FUNCTION_BLOCK "LAcycCom_WriteDriveParams"
{ S7_Optimized_Access := 'TRUE' }
AUTHOR : 'tech.team.motioncontrol@siemens.com'
FAMILY : AcycCom
VERSION : 1.5
   VAR_INPUT
      execute : Bool;
      parameterCount : Int := -1;
      driveObjectId { S7_HiddenAssignment := 'HideIfNoParamAssigned'} : Int := -1;
      hardwareId : HW_IO;
   END_VAR

   VAR_OUTPUT
      done { ExternalWritable := 'False'} : Bool;
      busy { ExternalWritable := 'False'} : Bool;
      error { ExternalWritable := 'False'} : Bool;
      status { ExternalWritable := 'False'} : Word := #STATUS_NO_CALL;
      diagnostics { ExternalWritable := 'False'} : "LAcycCom_typeDriveDiagnostics";
   END_VAR

   VAR_IN_OUT
      requestBuffer : "LAcycCom_typeRequestBuffer";
      dataset : Variant;
   END_VAR

   VAR
      statExecuteOld { ExternalAccessible := 'False'; ExternalVisible := 'False'; ExternalWritable := 'False'} : Bool := FALSE;
      statBusy { ExternalAccessible := 'False'; ExternalVisible := 'False'; ExternalWritable := 'False'} : Bool := FALSE;
      statDone { ExternalAccessible := 'False'; ExternalVisible := 'False'; ExternalWritable := 'False'} : Bool := FALSE;
      statError { ExternalAccessible := 'False'; ExternalVisible := 'False'; ExternalWritable := 'False'} : Bool := FALSE;
      statCmdBusy { ExternalAccessible := 'False'; ExternalVisible := 'False'; ExternalWritable := 'False'} : Bool := FALSE;
      statCmdDone { ExternalAccessible := 'False'; ExternalVisible := 'False'; ExternalWritable := 'False'} : Bool := FALSE;
      statCmdError { ExternalAccessible := 'False'; ExternalVisible := 'False'; ExternalWritable := 'False'} : Bool := FALSE;
      statTimerStart { ExternalAccessible := 'False'; ExternalVisible := 'False'; ExternalWritable := 'False'} : Bool := FALSE;
      statDoId { ExternalAccessible := 'False'; ExternalVisible := 'False'; ExternalWritable := 'False'} : Byte := 16#00;
      statHwId { ExternalAccessible := 'False'; ExternalVisible := 'False'; ExternalWritable := 'False'} : HW_IO := 16#0000;
      statRefNo { ExternalAccessible := 'False'; ExternalVisible := 'False'; ExternalWritable := 'False'} : Byte := 16#00;
      statStatus { ExternalAccessible := 'False'; ExternalVisible := 'False'; ExternalWritable := 'False'} : Word := #STATUS_NO_CALL;
      statSubfunctionStatus { ExternalAccessible := 'False'; ExternalVisible := 'False'; ExternalWritable := 'False'} : Word := 16#0000;
      statWithoutResourceManager { ExternalAccessible := 'False'; ExternalVisible := 'False'; ExternalWritable := 'False'} : Bool := FALSE;
      statFBState { ExternalAccessible := 'False'; ExternalVisible := 'False'; ExternalWritable := 'False'} : SInt := #FB_IDLE;
      statFBSubState { ExternalAccessible := 'False'; ExternalVisible := 'False'; ExternalWritable := 'False'} : SInt := #FB_BUSY_WRREC_1;
      statFBSubStateOld { ExternalAccessible := 'False'; ExternalVisible := 'False'; ExternalWritable := 'False'} : SInt := #FB_BUSY_WRREC_1;
      statStateNumber { ExternalAccessible := 'False'; ExternalVisible := 'False'; ExternalWritable := 'False'} : SInt := 0;
      statDatasetType { ExternalAccessible := 'False'; ExternalVisible := 'False'; ExternalWritable := 'False'} : SInt := 0;
      statErrorCount { ExternalAccessible := 'False'; ExternalVisible := 'False'; ExternalWritable := 'False'} : UInt := 16#0000;
      statAllocatedIndex { ExternalAccessible := 'False'; ExternalVisible := 'False'; ExternalWritable := 'False'} : Int := 0;
      statCountOfElements { ExternalAccessible := 'False'; ExternalVisible := 'False'; ExternalWritable := 'False'} : Int := 0;
      statFirstParameterError { ExternalAccessible := 'False'; ExternalVisible := 'False'; ExternalWritable := 'False'} : Int := -1;
      statWarningRetriggering { ExternalAccessible := 'False'; ExternalVisible := 'False'; ExternalWritable := 'False'} : Bool;
      statDataRecordNo { ExternalAccessible := 'False'; ExternalVisible := 'False'; ExternalWritable := 'False'} : DInt;
      statParameter { ExternalAccessible := 'False'; ExternalVisible := 'False'; ExternalWritable := 'False'} : Array[0..#WRITE_PARAMETERS_UPPER_LIM] of Struct
         parameterNo { ExternalAccessible := 'False'; ExternalVisible := 'False'; ExternalWritable := 'False'} : UInt;
         index { ExternalAccessible := 'False'; ExternalVisible := 'False'; ExternalWritable := 'False'} : UInt;
         realValue { ExternalAccessible := 'False'; ExternalVisible := 'False'; ExternalWritable := 'False'} : Real;
         dwordValue { ExternalAccessible := 'False'; ExternalVisible := 'False'; ExternalWritable := 'False'} : DWord;
         format { ExternalAccessible := 'False'; ExternalVisible := 'False'; ExternalWritable := 'False'} : Byte;
         errorValue { ExternalAccessible := 'False'; ExternalVisible := 'False'; ExternalWritable := 'False'} : Byte;
      END_STRUCT;
      statReqReadParameter { ExternalAccessible := 'False'; ExternalVisible := 'False'; ExternalWritable := 'False'} : Struct
         header { ExternalAccessible := 'False'; ExternalVisible := 'False'; ExternalWritable := 'False'} : Struct
            refNo { ExternalAccessible := 'False'; ExternalVisible := 'False'; ExternalWritable := 'False'} : Byte;
            reqId { ExternalAccessible := 'False'; ExternalVisible := 'False'; ExternalWritable := 'False'} : Byte;
            doId { ExternalAccessible := 'False'; ExternalVisible := 'False'; ExternalWritable := 'False'} : Byte;
            parameterNo { ExternalAccessible := 'False'; ExternalVisible := 'False'; ExternalWritable := 'False'} : Byte;
         END_STRUCT;
         parameterAddress { ExternalAccessible := 'False'; ExternalVisible := 'False'; ExternalWritable := 'False'} : Array[0..#WRITE_PARAMETERS_UPPER_LIM] of Struct
            attribute { ExternalAccessible := 'False'; ExternalVisible := 'False'; ExternalWritable := 'False'} : Byte;
            elementNo { ExternalAccessible := 'False'; ExternalVisible := 'False'; ExternalWritable := 'False'} : Byte;
            parameterNo { ExternalAccessible := 'False'; ExternalVisible := 'False'; ExternalWritable := 'False'} : UInt;
            index { ExternalAccessible := 'False'; ExternalVisible := 'False'; ExternalWritable := 'False'} : UInt;
         END_STRUCT;
      END_STRUCT;
      statReqParameterInit { ExternalAccessible := 'False'; ExternalVisible := 'False'; ExternalWritable := 'False'} : Struct
         attribute { ExternalAccessible := 'False'; ExternalVisible := 'False'; ExternalWritable := 'False'} : Byte := 16#10;
         elementNo { ExternalAccessible := 'False'; ExternalVisible := 'False'; ExternalWritable := 'False'} : Byte := 16#01;
         parameterNo { ExternalAccessible := 'False'; ExternalVisible := 'False'; ExternalWritable := 'False'} : UInt := 0;
         index { ExternalAccessible := 'False'; ExternalVisible := 'False'; ExternalWritable := 'False'} : UInt := 0;
      END_STRUCT;
      statReqWriteParameter { ExternalAccessible := 'False'; ExternalVisible := 'False'; ExternalWritable := 'False'} : Struct
         header { ExternalAccessible := 'False'; ExternalVisible := 'False'; ExternalWritable := 'False'} : Struct
            refNo { ExternalAccessible := 'False'; ExternalVisible := 'False'; ExternalWritable := 'False'} : Byte;
            reqId { ExternalAccessible := 'False'; ExternalVisible := 'False'; ExternalWritable := 'False'} : Byte;
            doId { ExternalAccessible := 'False'; ExternalVisible := 'False'; ExternalWritable := 'False'} : Byte;
            parameterNo { ExternalAccessible := 'False'; ExternalVisible := 'False'; ExternalWritable := 'False'} : Byte;
         END_STRUCT;
         data { ExternalAccessible := 'False'; ExternalVisible := 'False'; ExternalWritable := 'False'} : Array[0..#LENGTH_WRITE_TELEGRAM_UPPER_LIM] of Byte;
      END_STRUCT;
      statRespParameter { ExternalAccessible := 'False'; ExternalVisible := 'False'; ExternalWritable := 'False'} : Struct
         header { ExternalAccessible := 'False'; ExternalVisible := 'False'; ExternalWritable := 'False'} : Struct
            refNo { ExternalAccessible := 'False'; ExternalVisible := 'False'; ExternalWritable := 'False'} : Byte;
            reqId { ExternalAccessible := 'False'; ExternalVisible := 'False'; ExternalWritable := 'False'} : Byte;
            doId { ExternalAccessible := 'False'; ExternalVisible := 'False'; ExternalWritable := 'False'} : Byte;
            parameterNo { ExternalAccessible := 'False'; ExternalVisible := 'False'; ExternalWritable := 'False'} : Byte;
         END_STRUCT;
         data { ExternalAccessible := 'False'; ExternalVisible := 'False'; ExternalWritable := 'False'} : Array[0..#LENGTH_READ_TELEGRAM_UPPER_LIM] of Byte;
      END_STRUCT;
      instWRREC {InstructionName := 'WRREC'; LibVersion := '1.1'; ExternalAccessible := 'False'; ExternalVisible := 'False'; ExternalWritable := 'False'} : WRREC;
      instRDREC {InstructionName := 'RDREC'; LibVersion := '1.0'; ExternalAccessible := 'False'; ExternalVisible := 'False'; ExternalWritable := 'False'} : RDREC;
      instIECTimer {InstructionName := 'TON_TIME'; LibVersion := '1.0'; ExternalAccessible := 'False'; ExternalVisible := 'False'; ExternalWritable := 'False'} : TON_TIME;
   END_VAR

   VAR_TEMP
      tempExecute : Bool;
      tempCmdValid : Bool;
      tempStatusWord : Word;
      tempParameterCount : Int;
      tempPointer : Int;
      tempLoopIndex : Int;
      tempBlkVariant : Int;
      tempLastQueueElement : Int;
      tempCmdStatus : DWord;
      tempDWord : DWord;
      tempVoidDiagnostics : "LAcycCom_typeDriveDiagnostics";
      tempActualElementReal : "LAcycCom_typeDriveDatasetReal";
      tempActualElementDWord : "LAcycCom_typeDriveDatasetDWord";
      tempSilentOperationData : "LAcycCom_typeDriveSilentOperation";
      tempVoidHeader : Struct
         reqRef : Byte;
         reqId : Byte;
         axisNo : Byte;
         parameterNo : Byte;
      END_STRUCT;
      tempDatasetRealValue : Array[0..1] of "LAcycCom_typeDriveDatasetReal";
      tempDatasetDWordValue : Array[0..1] of "LAcycCom_typeDriveDatasetDWord";
   END_VAR

   VAR CONSTANT
      DATA_TYPE_SILENT : SInt := 1;
      DATA_TYPE_DATASET_REAL : SInt := 2;
      DATA_TYPE_DATASET_DWORD : SInt := 3;
      NO_PARAMETER_ERROR : Int := -1;
      ALL_ELEMENTS_OCCUPIED : Int := -1;
      FB_IDLE : SInt := 0;
      FB_FIRST_CYCLE : SInt := 1;
      FB_ALLOCATE : SInt := 2;
      FB_GET_RESOURCE : SInt := 3;
      FB_BUSY : SInt := 4;
      FB_RELEASE : SInt := 5;
      FB_DONE : SInt := 6;
      FB_ERROR : SInt := 7;
      FB_BUSY_WRREC_1 : SInt := 8;
      FB_BUSY_WRREC_2 : SInt := 9;
      FB_BUSY_RDREC_1 : SInt := 10;
      FB_BUSY_RDREC_2 : SInt := 11;
      FB_BUSY_WAIT : SInt := 12;
      FORMAT_INTEGER_8 : SInt := 2;
      FORMAT_INTEGER_16 : SInt := 3;
      FORMAT_INTEGER_32 : SInt := 4;
      FORMAT_UNSIGNED_8 : SInt := 5;
      FORMAT_UNSIGNED_16 : SInt := 6;
      FORMAT_UNSIGNED_32 : SInt := 7;
      FORMAT_FLOATING_POINT : SInt := 8;
      FORMAT_OCTET_STRING : SInt := 10;
      FORMAT_TIME_DIFFERENCE : SInt := 13;
      FORMAT_ZERO : SInt := 64;
      FORMAT_BYTE : SInt := 65;
      FORMAT_WORD : SInt := 66;
      FORMAT_DOUBLE_WORD : SInt := 67;
      FORMAT_ERROR : Byte := 16#44;
      WRITE_PARAMETERS_UPPER_LIM : Int := 18;
      SILENT_OPERATION_PARA_UPPER_LIM : Int := 17;
      LENGTH_WRITE_TELEGRAM_UPPER_LIM : Int := 227;
      LENGTH_READ_TELEGRAM_UPPER_LIM : Int := 113;
      MAX_ERROR_COUNT : UInt := 100;
      TIMER_TEMP_ERROR : Time := T#200MS;
      TIMER_ALLOCATION : Time := T#10S;
      MAX_DRIVE_OBJECT_NO : Int := 254;
      STATUS_EXECUTION_FINISHED : Word := 16#0000;
      STATUS_NO_CALL : Word := 16#7000;
      STATUS_ALLOCATE : Word := 16#7001;
      STATUS_GET_RESOURCE : Word := 16#7002;
      STATUS_BUSY : Word := 16#7003;
      STATUS_RELEASE : Word := 16#7004;
      WARN_EXECUTE : Word := 16#7100;
      WARN_EXECUTE_SET_DURING_PROCESSING : Word := 16#7101;
      ERR_NO_OF_PARAMETERS : Word := 16#8001;
      ERR_REQUEST_REJECTED : Word := 16#8004;
      ERR_RESOURCE_RELEASED : Word := 16#8005;
      ERR_AMBIGUOUS_FB_CALL : Word := 16#8006;
      ERR_INVALID_DATA_TYPE : Word := 16#8200;
      ERR_INVALID_BUF_INDEX : Word := 16#8201;
      ERR_INVALID_DRIVE_OBJECT_ID : Word := 16#8208;
      ERR_COMMAND_TIMEOUT : Word := 16#8600;
      ERR_RDREC_TEMP_COUNTER : Word := 16#8601;
      ERR_WRREC_TEMP_COUNTER : Word := 16#8602;
      ERR_WRREC : Word := 16#8603;
      ERR_RDREC : Word := 16#8604;
      ERR_REFERENCE_NO : Word := 16#8605;
      ERR_RESPONSE_ID : Word := 16#8606;
      ERR_PARAMETER_NO : Word := 16#8607;
      ERR_DRIVE_OBJECT_NO : Word := 16#8608;
      ERR_ALLOCATION_TIME : Word := 16#8609;
      ERR_MOVE_BLK_VARIANT : Word := 16#8610;
      ERR_UNDEFINED_STATE : Word := 16#8611;
      ERR_UNDEFINED_SUBSTATE : Word := 16#8612;
      ERR_PARAMETER : Word := 16#8619;
   END_VAR


BEGIN
	//==========================================================================================
	// SIEMENS AG
	// (c)Copyright 2020 All Rights Reserved
	//------------------------------------------------------------------------------------------
	// Library: LAcycCom
	// Tested with: S7-1513-1 PN
	// Engineering: TIA Portal V15
	// Restrictions: ---
	// Requirements: S7-1200/1500
	//               FB LAcycCom_ResourceManager is required
	// Functionality: Writes parameters into a drive object according to the configured dataset
	//------------------------------------------------------------------------------------------
	// Change log table:
	// Version    Date          Expert in charge    Changes applied
	// 01.00.00   05.05.2015    AW                  release
	// 01.01.00   27.01.2016    AW                  values of MAX_ERROR_COUNT and TIMER_TEMP_ERROR changed
	// 01.03.00   05.07.2016    AL                  output added: diagnostics.status
	//                                              bugfix error handling (if execute input is set only for 1 cycle)
	// 01.03.01   21.11.2016    AL                  prevent reentrant calls (added warning #WARN_EXECUTE_SET_DURING_PROCESSING
	//                                                                       and error #ERR_AMBIGUOUS_FB_CALL)
	// 01.03.02   22.11.2017    AL                  added handling of error 80A0 (RDREC)
	//                                              added handling of error 80A1 (WRREC)
	//                                              added errorValue to "LAcycCom_typeDriveDiagnostics"
	// 01.03.03   13.03.2018    AL                  values of MAX_ERROR_COUNT and TIMER_TEMP_ERROR changed
	// 01.05.00   31.10.2018    AL                  added support of Base Mode Parameter Access local (16#B02E)
	//                                              (driveObjectId < 0: local, driveObjectId >= 0: Base Mode Parameter Access global via dataset 47)
	//                                              input 'driveObjectId' data type changed from USInt to Int
	//                                              changed handling of OCTET_STRING format
	// 01.05.01   11.10.2019    AL                  bugfix lockBuffer
	//                                              value of MAX_ERROR_COUNT changed
	// 01.05.02   19.05.2020    CR                  new errorId when input 'driveObjectId' is out of range
	//
	//------------------------------------------------------------------------------------------
	// Function block: LAcycCom_WriteDriveParams
	//===========================================================================================
	//

	//----------------------------------------------------------------------
	// Determine which PLC data type for writeDataset is in use
	//----------------------------------------------------------------------
	IF (TypeOf(#dataset) = TypeOf(#tempDatasetRealValue)) OR (TypeOf(#dataset) = TypeOf(#tempDatasetDWordValue)) THEN
	  #tempExecute := #execute;

	ELSIF (TypeOf(#dataset) = LAcycCom_typeDriveSilentOperation) THEN
	  #tempBlkVariant := MOVE_BLK_VARIANT(SRC := #dataset, COUNT := 1, SRC_INDEX := 0, DEST_INDEX := 0, DEST => #tempSilentOperationData);

	  // Error occurred during MOVE_BLK_VARIANT command
	  IF (#tempBlkVariant <> 0) THEN
	    #statError := TRUE;
	    #statStateNumber := #statFBState;
	    #statSubfunctionStatus := INT_TO_WORD(#tempBlkVariant);
	    #statStatus := #ERR_MOVE_BLK_VARIANT;
	    #statFBState := #FB_ERROR;
	  END_IF;

	  #tempExecute := #tempSilentOperationData.functionBlockCommand.%X1;

	  // Input execute is set during silent operation
	  IF (#execute = TRUE) AND (#statError = FALSE) THEN
	    #statStatus := #WARN_EXECUTE;
	    #diagnostics.status := #statStatus;
	  END_IF;

	ELSE
	  #statError := TRUE;
	  #statStateNumber := #statFBState;
	  #statStatus := #ERR_INVALID_DATA_TYPE;
	  #statFBState := #FB_ERROR;
	END_IF;

	//----------------------------------------------------------------------
	// Processing
	//----------------------------------------------------------------------
	// Rising edge of execute starts functionality
	IF (#tempExecute = TRUE) AND (#statExecuteOld = FALSE) AND (#statBusy = TRUE) THEN
	  // Input execute is set during processing
	  #statStatus := #WARN_EXECUTE_SET_DURING_PROCESSING;
	  #statWarningRetriggering := TRUE;

	ELSIF (#tempExecute = TRUE) AND (#statExecuteOld = FALSE) THEN
	  // First call
	  // Initialisation
	  #statDone := FALSE;
	  #statBusy := TRUE;
	  #statError := FALSE;
	  #statCountOfElements := 0;
	  #statAllocatedIndex := 0;
	  #statHwId := 16#0;
	  #statSubfunctionStatus := 16#0;
	  #statDoId := 0;
	  #statDataRecordNo := 0;
	  #statStateNumber := 0;
	  #statFirstParameterError := -1;
	  #statCmdBusy := FALSE;
	  #statCmdDone := FALSE;
	  #statCmdError := FALSE;
	  #statErrorCount := 0;
	  #statWarningRetriggering := FALSE;
	  #statFBSubState := #FB_BUSY_WRREC_1;
	  #statFBState := #FB_FIRST_CYCLE;

	  #instIECTimer(IN := FALSE,
	                PT := #TIMER_ALLOCATION);

	  // FB is currently inactive
	ELSIF (#tempExecute = FALSE) AND (#statBusy = FALSE)
	THEN
	  #statError := FALSE;
	  #statBusy := FALSE;
	  #statDone := FALSE;
	  #statFBState := #FB_IDLE;

	  IF (#statStatus = #WARN_EXECUTE) AND (#execute = FALSE) OR (#statStatus <> #WARN_EXECUTE) THEN
	    #statStatus := #STATUS_NO_CALL;
	  END_IF;
	END_IF; // #tempExecute AND NOT #statExecuteOld

	//----------------------------------------------------------------------
	// State Machine
	//----------------------------------------------------------------------

	IF (#statBusy = TRUE) AND (#statError = FALSE) THEN  // Functionality running
	  CASE #statFBState OF
	    #FB_FIRST_CYCLE:  // First cycle state

	      // Determine which PLC data type for readDataset is in use
	      IF (TypeOf(#dataset) = TypeOf(#tempDatasetRealValue)) THEN
	        #statDatasetType := #DATA_TYPE_DATASET_REAL;

	      ELSIF (TypeOf(#dataset) = TypeOf(#tempDatasetDWordValue)) THEN
	        #statDatasetType := #DATA_TYPE_DATASET_DWORD;

	      ELSIF (TypeOf(#dataset) = LAcycCom_typeDriveSilentOperation) THEN
	        #statDatasetType := #DATA_TYPE_SILENT;
	      END_IF;

	      // Clearing the dataset in silent operation mode
	      FOR #tempLoopIndex := 0 TO #SILENT_OPERATION_PARA_UPPER_LIM DO
	        #tempSilentOperationData.dataset[#tempLoopIndex].errorValue := 16#FF;
	      END_FOR;

	      // Clearing the sending read buffer
	      #statReqReadParameter.header := #tempVoidHeader;
	      FOR #tempLoopIndex := 0 TO #WRITE_PARAMETERS_UPPER_LIM DO
	        #statReqReadParameter.parameterAddress[#tempLoopIndex] := #statReqParameterInit;
	      END_FOR;

	      // Clearing the sending write buffer
	      #statReqWriteParameter.header := #tempVoidHeader;
	      FOR #tempLoopIndex := 0 TO #LENGTH_WRITE_TELEGRAM_UPPER_LIM DO
	        #statReqWriteParameter.data[#tempLoopIndex] := 16#00;
	      END_FOR;

	      // Clearing the receive buffer
	      #statRespParameter.header := #tempVoidHeader;
	      FOR #tempLoopIndex := 0 TO #LENGTH_READ_TELEGRAM_UPPER_LIM DO
	        #statRespParameter.data[#tempLoopIndex] := 16#00;
	      END_FOR;

	      // Initialization after start, depending on the used PLC data type
	      IF (#statDatasetType = #DATA_TYPE_DATASET_REAL) OR (#statDatasetType = #DATA_TYPE_DATASET_DWORD) THEN
	        IF #driveObjectId < 0 THEN // V1.5
	          #statDataRecordNo := 16#B02E; // Base Mode Parameter Access local; doId not relevant
	          #statDoId := 0;

	        ELSIF (#driveObjectId <= #MAX_DRIVE_OBJECT_NO)
	          AND (#driveObjectId <> 0)
	        THEN // V1.5.2
	          #statDataRecordNo := 47; // Data record 47; Base Mode Parameter Access global
	          #statDoId := INT_TO_BYTE(#driveObjectId);

	        ELSE // V1.5.2
	          // Wrong drive object ID at input
	          #statError := TRUE;
	          #statStateNumber := #statFBState;
	          #statStatus := #ERR_INVALID_DRIVE_OBJECT_ID;
	          #statFBState := #FB_ERROR;
	        END_IF;

	        #statHwId := #hardwareId;
	        #tempParameterCount := #parameterCount;
	      ELSE
	        IF #tempSilentOperationData.driveObjectId < 0 THEN // V1.5
	          #statDataRecordNo := 16#B02E; // Base Mode Parameter Access local; doId not relevant
	          #statDoId := 0;
	        ELSE
	          #statDataRecordNo := 47; // Data record 47; Base Mode Parameter Access global
	          #statDoId := INT_TO_BYTE(#tempSilentOperationData.driveObjectId);
	        END_IF;
	        #statHwId := #tempSilentOperationData.hardwareId;
	        #tempParameterCount := #tempSilentOperationData.parameterCount;
	      END_IF;

	      #diagnostics := #tempVoidDiagnostics;
	      // Input execute is set during silent operation
	      IF #statStatus = #WARN_EXECUTE THEN
	        #diagnostics.status := #statStatus;
	      END_IF;
	      #diagnostics.driveObjectId := #statDoId;
	      #diagnostics.hardwareId := #statHwId;
	      #diagnostics.firstParameterError := #statFirstParameterError; // V1.3.2
	      #diagnostics.errorValue := 16#FF; // V1.3.2

	      // Reference number for next request
	      #statRefNo := #statRefNo + 1;

	      IF #statError THEN // V1.5.2: Check if error appeared
	        ;

	      // Next state is depending on the FB mode
	      ELSIF (#statWithoutResourceManager = FALSE) THEN
	        #statStatus := #STATUS_ALLOCATE;
	        #statFBState := #FB_ALLOCATE;

	      ELSE
	        #statStatus := #STATUS_BUSY;
	        #statFBState := #FB_BUSY;
	        #statFBSubState := #FB_BUSY_WRREC_1;
	      END_IF; // #statMode = #MODE_WITH_BUFFER_MANAGER

	      // Calculates the amount of parameters (only if no error occurs)
	      IF (#statError = FALSE) THEN
	        IF (#statDatasetType = #DATA_TYPE_SILENT) THEN
	          // Check if 0 < parameterCount <= 18
	          IF (#tempParameterCount > 0) AND (#tempParameterCount <= #SILENT_OPERATION_PARA_UPPER_LIM + 1) THEN
	            #statCountOfElements := #tempParameterCount;
	            #diagnostics.parameterCount := #statCountOfElements;

	          ELSE
	            #statError := TRUE;
	            #statStateNumber := #statFBState;
	            #statStatus := #ERR_NO_OF_PARAMETERS;
	            #statFBState := #FB_ERROR;
	          END_IF; // #tempParameterCount <= #MAX_NO_OF_PARAMETERS

	        ELSE
	          // Calculates the count of elements in readDataset if numberOfParameters < 1
	          IF (#tempParameterCount < 1) AND
	            (CountOfElements(#dataset) <= #WRITE_PARAMETERS_UPPER_LIM + 1) AND
	            ("LACYCCOM_WRITE_PARAMETERS_UPPER_LIM" <= #WRITE_PARAMETERS_UPPER_LIM)
	          THEN
	            #statCountOfElements := UDINT_TO_INT(CountOfElements(#dataset));
	            #diagnostics.parameterCount := #statCountOfElements;

	          ELSIF (#tempParameterCount >= 1) AND // V1.3.2
	            // Check if numberOfParameters <= 19
	            (#tempParameterCount <= #WRITE_PARAMETERS_UPPER_LIM + 1) AND
	            (CountOfElements(#dataset) >= #tempParameterCount) AND
	            ("LACYCCOM_WRITE_PARAMETERS_UPPER_LIM" <= #WRITE_PARAMETERS_UPPER_LIM)
	          THEN
	            #statCountOfElements := #tempParameterCount;
	            #diagnostics.parameterCount := #statCountOfElements;

	          ELSE
	            #statError := TRUE;
	            #statStateNumber := #statFBState;
	            #statStatus := #ERR_NO_OF_PARAMETERS;
	            #statFBState := #FB_ERROR;
	          END_IF;
	        END_IF; // #tempDatasetType = #DATA_TYPE_SILENT
	      END_IF;

	    #FB_ALLOCATE:

	      // Allocation of a request element
	      IF (#requestBuffer.header.lockBuffer = FALSE) AND (#requestBuffer.header.nextFreeElement >= 0) AND (#requestBuffer.header.nextFreeElement <= "LACYCCOM_BUFFER_ELEMENTS_UPPER_LIM") THEN
	        #requestBuffer.header.lockBuffer := TRUE;
	        #statAllocatedIndex := #requestBuffer.header.nextFreeElement;
	        #requestBuffer.elements[#statAllocatedIndex].state := 16#00;
	        #requestBuffer.elements[#statAllocatedIndex].state.%X0 := TRUE;
	        #requestBuffer.elements[#statAllocatedIndex].hardwareId := #statHwId;
	        #requestBuffer.elements[#statAllocatedIndex].queueElementNext := -1;
	        #statTimerStart := FALSE;
	        #statStatus := #STATUS_GET_RESOURCE;
	        #statFBState := #FB_GET_RESOURCE;

	        // Build up queue
	        IF (#requestBuffer.header.firstQueueElement >= 0) THEN
	          // Find last queue element
	          #tempLoopIndex := #requestBuffer.header.firstQueueElement;
	          WHILE (#tempLoopIndex >= 0) DO
	            #tempLastQueueElement := #tempLoopIndex;
	            #tempLoopIndex := #requestBuffer.elements[#tempLoopIndex].queueElementNext;
	          END_WHILE;

	          // Insert into list after last element
	          #requestBuffer.elements[#tempLastQueueElement].queueElementNext := #statAllocatedIndex;
	          #requestBuffer.elements[#statAllocatedIndex].queueElementPrevious := #tempLastQueueElement;
	        ELSE
	          // Element is first element in queue
	          #requestBuffer.header.firstQueueElement := #statAllocatedIndex;
	          #requestBuffer.elements[#statAllocatedIndex].queueElementPrevious := -1;
	        END_IF;

	        // Searching for the next free request element
	        FOR #tempLoopIndex := 0 TO "LACYCCOM_BUFFER_ELEMENTS_UPPER_LIM" DO
	          IF (#requestBuffer.elements[#tempLoopIndex].state.%X0 = FALSE) THEN
	            #requestBuffer.header.nextFreeElement := #tempLoopIndex;
	            EXIT;
	          END_IF;

	          // All request elements are occupied
	          IF (#tempLoopIndex = "LACYCCOM_BUFFER_ELEMENTS_UPPER_LIM") THEN
	            #requestBuffer.header.nextFreeElement := #ALL_ELEMENTS_OCCUPIED;
	          END_IF;
	        END_FOR;

	        #requestBuffer.header.lockBuffer := FALSE;

	      ELSIF (#instIECTimer.Q = TRUE) THEN
	        #statError := TRUE;
	        #statStateNumber := #statFBState;
	        #statStatus := #ERR_ALLOCATION_TIME;
	        #statFBState := #FB_ERROR;

	      ELSE
	        ; // Waiting until lockbit is reset and a request element is available
	      END_IF; // (#buffer.lockBuffer = FALSE) AND (#buffer.actualWriteIndex >= 0)

	      #instIECTimer(IN := #statTimerStart,
	                    PT := #TIMER_ALLOCATION);

	      #statTimerStart := TRUE;
	      IF (#instIECTimer.Q = TRUE) THEN
	        #statTimerStart := FALSE;
	      END_IF;

	    #FB_GET_RESOURCE:

	      // Check buffer index for correctness
	      IF (#statAllocatedIndex < 0) OR (#statAllocatedIndex > "LACYCCOM_BUFFER_ELEMENTS_UPPER_LIM") THEN
	        #statError := TRUE;
	        #statStateNumber := #statFBState;
	        #statStatus := #ERR_INVALID_BUF_INDEX;
	        #statFBState := #FB_ERROR;

	      ELSE
	        IF (#requestBuffer.elements[#statAllocatedIndex].state.%X0 = FALSE) OR
	          (#requestBuffer.elements[#statAllocatedIndex].state.%X3 = TRUE)
	        THEN
	          // Request was rejected by buffer manager
	          #statError := TRUE;
	          #statStateNumber := #statFBState;
	          #statStatus := #ERR_REQUEST_REJECTED;
	          #statFBState := #FB_ERROR;

	        ELSIF (#requestBuffer.elements[#statAllocatedIndex].state.%X2 = TRUE) THEN
	          // Request already released
	          #statError := TRUE;
	          #statStateNumber := #statFBState;
	          #statStatus := #ERR_RESOURCE_RELEASED;
	          #statFBState := #FB_ERROR;

	        ELSIF (#requestBuffer.elements[#statAllocatedIndex].state.%X1 = TRUE) THEN
	          // Element is enabled
	          #statStatus := #STATUS_BUSY;
	          #statFBState := #FB_BUSY;
	          #statFBSubState := #FB_BUSY_WRREC_1;

	        ELSE
	          // Element not enabled yet
	          //
	          #statStatus := #STATUS_GET_RESOURCE;
	        END_IF;

	      END_IF;

	    #FB_BUSY:

	      IF ((#requestBuffer.elements[#statAllocatedIndex].state.%X1 = TRUE) AND (#statWithoutResourceManager = FALSE)
	        AND (#requestBuffer.elements[#statAllocatedIndex].state.%X3 = FALSE)) OR (#statWithoutResourceManager = TRUE)
	      THEN

	        CASE #statFBSubState OF
	          #FB_BUSY_WRREC_1, #FB_BUSY_WRREC_2:  // Writing the dataset configuration into the drive object

	            IF (#statCmdBusy = FALSE) AND (#statFBSubState = #FB_BUSY_WRREC_1) AND (#statError = FALSE) THEN
	              // Resets WRREC command
	              #instWRREC(REQ := FALSE);

	              // Creating header data
	              #statReqReadParameter.header.refNo := #statRefNo; // Telegram reference number
	              #statReqReadParameter.header.reqId := 16#01;  // 0x01 = request parameters
	              #statReqReadParameter.header.doId := #statDoId;  // Drive object identification number
	              #statReqReadParameter.header.parameterNo := INT_TO_BYTE(#statCountOfElements);  // Count of parameters

	              // Copying the dataset into a static variable (depending on the used PLC data type)
	              IF (#statDatasetType = #DATA_TYPE_SILENT) THEN
	                FOR #tempLoopIndex := 0 TO #statCountOfElements - 1 BY 1 DO
	                  #statParameter[#tempLoopIndex].index := 0;
	                  #statParameter[#tempLoopIndex].parameterNo := #tempSilentOperationData.dataset[#tempLoopIndex].parameterNumber;
	                  #statParameter[#tempLoopIndex].realValue := #tempSilentOperationData.dataset[#tempLoopIndex].value;
	                  #statReqReadParameter.parameterAddress[#tempLoopIndex].parameterNo := #statParameter[#tempLoopIndex].parameterNo;  // Parameter number
	                  #statReqReadParameter.parameterAddress[#tempLoopIndex].index := #statParameter[#tempLoopIndex].index;  // Subindex of parameter
	                END_FOR;

	              ELSIF (#statDatasetType = #DATA_TYPE_DATASET_REAL) THEN
	                FOR #tempLoopIndex := 0 TO #statCountOfElements - 1 BY 1 DO
	                  #tempBlkVariant := MOVE_BLK_VARIANT(SRC := #dataset, COUNT := 1, SRC_INDEX := #tempLoopIndex, DEST_INDEX := 0, DEST => #tempActualElementReal);

	                  // Error occurred during MOVE_BLK_VARIANT command
	                  IF (#tempBlkVariant <> 0) THEN
	                    #statError := TRUE;
	                    #statStateNumber := #statFBSubState;
	                    #statSubfunctionStatus := INT_TO_WORD(#tempBlkVariant);
	                    #statStatus := #ERR_MOVE_BLK_VARIANT;
	                    #statFBState := #FB_ERROR;
	                    #diagnostics.firstParameterError := #tempLoopIndex;
	                    EXIT;
	                  END_IF;

	                  #statParameter[#tempLoopIndex].index := 0;
	                  #statParameter[#tempLoopIndex].parameterNo := #tempActualElementReal.parameterNumber;
	                  #statParameter[#tempLoopIndex].realValue := #tempActualElementReal.value;
	                  #statReqReadParameter.parameterAddress[#tempLoopIndex].parameterNo := #statParameter[#tempLoopIndex].parameterNo;  // Parameter number
	                  #statReqReadParameter.parameterAddress[#tempLoopIndex].index := #statParameter[#tempLoopIndex].index;  // Subindex of parameter
	                END_FOR;

	                // If #DATA_TYPE_DATASET_DWORD is in use
	              ELSE
	                FOR #tempLoopIndex := 0 TO #statCountOfElements - 1 BY 1 DO
	                  #tempBlkVariant := MOVE_BLK_VARIANT(SRC := #dataset, COUNT := 1, SRC_INDEX := #tempLoopIndex, DEST_INDEX := 0, DEST => #tempActualElementDWord);

	                  // Error occurred during MOVE_BLK_VARIANT command
	                  IF (#tempBlkVariant <> 0) THEN
	                    #statError := TRUE;
	                    #statStateNumber := #statFBSubState;
	                    #statSubfunctionStatus := INT_TO_WORD(#tempBlkVariant);
	                    #statStatus := #ERR_MOVE_BLK_VARIANT;
	                    #statFBState := #FB_ERROR;
	                    #diagnostics.firstParameterError := #tempLoopIndex;
	                    EXIT;
	                  END_IF;

	                  #statParameter[#tempLoopIndex].index := 0;
	                  #statParameter[#tempLoopIndex].parameterNo := #tempActualElementDWord.parameterNumber;
	                  #statParameter[#tempLoopIndex].dwordValue := #tempActualElementDWord.value;
	                  #statReqReadParameter.parameterAddress[#tempLoopIndex].parameterNo := #statParameter[#tempLoopIndex].parameterNo;  // Parameter number
	                  #statReqReadParameter.parameterAddress[#tempLoopIndex].index := #statParameter[#tempLoopIndex].index;  // Subindex of parameter
	                END_FOR;
	              END_IF;

	            ELSIF (#statCmdBusy = FALSE) AND (#statFBSubState = #FB_BUSY_WRREC_2) AND (#statError = FALSE) THEN
	              // Resets WRREC command
	              #instWRREC(REQ := FALSE);

	              #tempPointer := 0;
	              // Creating header data
	              #statReqWriteParameter.header.refNo := #statRefNo; // Telegram reference number
	              #statReqWriteParameter.header.reqId := 16#02;  // 0x02 = change parameters
	              #statReqWriteParameter.header.doId := #statDoId;  // Drive object identification number
	              #statReqWriteParameter.header.parameterNo := INT_TO_BYTE(#statCountOfElements);  // Count of parameters

	              FOR #tempLoopIndex := 0 TO #statCountOfElements - 1 BY 1 DO
	                #statReqWriteParameter.data[#tempPointer] := 16#10; // Attribute of parameters (0x10=Value, 0x30=Text)
	                #statReqWriteParameter.data[#tempPointer + 1] := 16#01; // No. of elements (for single elements=1)

	                IF (#statDatasetType = #DATA_TYPE_SILENT) THEN
	                  #statParameter[#tempLoopIndex].index := #tempSilentOperationData.dataset[#tempLoopIndex].index;
	                  #statParameter[#tempLoopIndex].parameterNo := #tempSilentOperationData.dataset[#tempLoopIndex].parameterNumber;

	                ELSIF (#statDatasetType = #DATA_TYPE_DATASET_REAL) THEN
	                  #tempBlkVariant := MOVE_BLK_VARIANT(SRC := #dataset, COUNT := 1, SRC_INDEX := #tempLoopIndex, DEST_INDEX := 0, DEST => #tempActualElementReal);

	                  // Error occurred during MOVE_BLK_VARIANT command
	                  IF (#tempBlkVariant <> 0) THEN
	                    #statError := TRUE;
	                    #statStateNumber := #statFBSubState;
	                    #statSubfunctionStatus := INT_TO_WORD(#tempBlkVariant);
	                    #statStatus := #ERR_MOVE_BLK_VARIANT;
	                    #statFBState := #FB_ERROR;
	                    #diagnostics.firstParameterError := #tempLoopIndex;
	                  END_IF;

	                  #statParameter[#tempLoopIndex].index := #tempActualElementReal.index;
	                  #statParameter[#tempLoopIndex].parameterNo := #tempActualElementReal.parameterNumber;

	                ELSE
	                  #tempBlkVariant := MOVE_BLK_VARIANT(SRC := #dataset, COUNT := 1, SRC_INDEX := #tempLoopIndex, DEST_INDEX := 0, DEST => #tempActualElementDWord);

	                  // Error occurred during MOVE_BLK_VARIANT command
	                  IF (#tempBlkVariant <> 0) THEN
	                    #statError := TRUE;
	                    #statStateNumber := #statFBSubState;
	                    #statSubfunctionStatus := INT_TO_WORD(#tempBlkVariant);
	                    #statStatus := #ERR_MOVE_BLK_VARIANT;
	                    #statFBState := #FB_ERROR;
	                    #diagnostics.firstParameterError := #tempLoopIndex;
	                  END_IF;

	                  #statParameter[#tempLoopIndex].index := #tempActualElementDWord.index;
	                  #statParameter[#tempLoopIndex].parameterNo := #tempActualElementDWord.parameterNumber;
	                END_IF;

	                // Parameter number
	                #statReqWriteParameter.data[#tempPointer + 3] := #statParameter[#tempLoopIndex].parameterNo.%B0;
	                #statReqWriteParameter.data[#tempPointer + 2] := #statParameter[#tempLoopIndex].parameterNo.%B1;

	                // Subindex of parameter
	                #statReqWriteParameter.data[#tempPointer + 5] := #statParameter[#tempLoopIndex].index.%B0;
	                #statReqWriteParameter.data[#tempPointer + 4] := #statParameter[#tempLoopIndex].index.%B1;

	                // Points to the next parameter address
	                #tempPointer := #tempPointer + 6;
	              END_FOR;

	              // Creating parameter address
	              FOR #tempLoopIndex := 0 TO #statCountOfElements - 1 BY 1 DO

	                IF (#statParameter[#tempLoopIndex].format = #FORMAT_ERROR) THEN
	                  #statParameter[#tempLoopIndex].format := SINT_TO_BYTE(#FORMAT_FLOATING_POINT);
	                END_IF;

	                #statReqWriteParameter.data[#tempPointer] := #statParameter[#tempLoopIndex].format; // Format of parameter
	                #statReqWriteParameter.data[#tempPointer + 1] := 16#01; // Count of values

	                CASE BYTE_TO_SINT(#statParameter[#tempLoopIndex].format) OF
	                  #FORMAT_INTEGER_8:
	                    IF (#statDatasetType = #DATA_TYPE_DATASET_REAL) OR (#statDatasetType = #DATA_TYPE_SILENT) THEN
	                      #tempDWord := SINT_TO_DWORD(REAL_TO_SINT(#statParameter[#tempLoopIndex].realValue));

	                    ELSE
	                      #tempDWord := #statParameter[#tempLoopIndex].dwordValue;
	                    END_IF;

	                    #statReqWriteParameter.data[#tempPointer + 3] := #tempDWord.%B1;
	                    #statReqWriteParameter.data[#tempPointer + 2] := #tempDWord.%B0;
	                    #tempPointer := #tempPointer + 4;  // Points to the next parameter address

	                  #FORMAT_INTEGER_16:
	                    IF (#statDatasetType = #DATA_TYPE_DATASET_REAL) OR (#statDatasetType = #DATA_TYPE_SILENT) THEN
	                      #tempDWord := DINT_TO_DWORD(REAL_TO_DINT(#statParameter[#tempLoopIndex].realValue));

	                    ELSE
	                      #tempDWord := #statParameter[#tempLoopIndex].dwordValue;
	                    END_IF;

	                    #statReqWriteParameter.data[#tempPointer + 3] := #tempDWord.%B0;
	                    #statReqWriteParameter.data[#tempPointer + 2] := #tempDWord.%B1;
	                    #tempPointer := #tempPointer + 4;  // Points to the next parameter address

	                  #FORMAT_INTEGER_32:
	                    IF (#statDatasetType = #DATA_TYPE_DATASET_REAL) OR (#statDatasetType = #DATA_TYPE_SILENT) THEN
	                      #tempDWord := DINT_TO_DWORD(REAL_TO_DINT(#statParameter[#tempLoopIndex].realValue));

	                    ELSE
	                      #tempDWord := #statParameter[#tempLoopIndex].dwordValue;
	                    END_IF;

	                    #statReqWriteParameter.data[#tempPointer + 5] := #tempDWord.%B0;
	                    #statReqWriteParameter.data[#tempPointer + 4] := #tempDWord.%B1;
	                    #statReqWriteParameter.data[#tempPointer + 3] := #tempDWord.%B2;
	                    #statReqWriteParameter.data[#tempPointer + 2] := #tempDWord.%B3;

	                    #tempPointer := #tempPointer + 6; // Points to the next parameter address

	                  #FORMAT_UNSIGNED_8, #FORMAT_OCTET_STRING: // V1.5 change OCTET_STRING:
	                    IF (#statDatasetType = #DATA_TYPE_DATASET_REAL) OR (#statDatasetType = #DATA_TYPE_SILENT) THEN
	                      #tempDWord := USINT_TO_DWORD(REAL_TO_USINT(#statParameter[#tempLoopIndex].realValue));

	                    ELSE
	                      #tempDWord := #statParameter[#tempLoopIndex].dwordValue;
	                    END_IF;

	                    #statReqWriteParameter.data[#tempPointer + 3] := #tempDWord.%B1;
	                    #statReqWriteParameter.data[#tempPointer + 2] := #tempDWord.%B0;
	                    #tempPointer := #tempPointer + 4;  // Points to the next parameter address

	                  #FORMAT_UNSIGNED_16:
	                    IF (#statDatasetType = #DATA_TYPE_DATASET_REAL) OR (#statDatasetType = #DATA_TYPE_SILENT) THEN
	                      #tempDWord := UDINT_TO_DWORD(REAL_TO_UDINT(#statParameter[#tempLoopIndex].realValue));

	                    ELSE
	                      #tempDWord := #statParameter[#tempLoopIndex].dwordValue;
	                    END_IF;

	                    #statReqWriteParameter.data[#tempPointer + 3] := #tempDWord.%B0;
	                    #statReqWriteParameter.data[#tempPointer + 2] := #tempDWord.%B1;
	                    #tempPointer := #tempPointer + 4;  // Points to the next parameter address

	                  #FORMAT_UNSIGNED_32, #FORMAT_TIME_DIFFERENCE:
	                    IF (#statDatasetType = #DATA_TYPE_DATASET_REAL) OR (#statDatasetType = #DATA_TYPE_SILENT) THEN
	                      #tempDWord := UDINT_TO_DWORD(REAL_TO_UDINT(#statParameter[#tempLoopIndex].realValue));

	                    ELSE
	                      #tempDWord := #statParameter[#tempLoopIndex].dwordValue;
	                    END_IF;

	                    #statReqWriteParameter.data[#tempPointer + 5] := #tempDWord.%B0;
	                    #statReqWriteParameter.data[#tempPointer + 4] := #tempDWord.%B1;
	                    #statReqWriteParameter.data[#tempPointer + 3] := #tempDWord.%B2;
	                    #statReqWriteParameter.data[#tempPointer + 2] := #tempDWord.%B3;

	                    #tempPointer := #tempPointer + 6; // Points to the next parameter address
	                  #FORMAT_FLOATING_POINT, #FORMAT_DOUBLE_WORD:
	                    IF (#statDatasetType = #DATA_TYPE_DATASET_REAL) OR (#statDatasetType = #DATA_TYPE_SILENT) THEN
	                      #tempDWord := REAL_TO_DWORD(#statParameter[#tempLoopIndex].realValue);

	                    ELSE
	                      #tempDWord := #statParameter[#tempLoopIndex].dwordValue;
	                    END_IF;

	                    #statReqWriteParameter.data[#tempPointer + 5] := #tempDWord.%B0;
	                    #statReqWriteParameter.data[#tempPointer + 4] := #tempDWord.%B1;
	                    #statReqWriteParameter.data[#tempPointer + 3] := #tempDWord.%B2;
	                    #statReqWriteParameter.data[#tempPointer + 2] := #tempDWord.%B3;

	                    #tempPointer := #tempPointer + 6;  // Points to the next parameter address
	                  #FORMAT_BYTE:
	                    IF (#statDatasetType = #DATA_TYPE_DATASET_REAL) OR (#statDatasetType = #DATA_TYPE_SILENT) THEN
	                      #tempDWord := REAL_TO_DWORD(#statParameter[#tempLoopIndex].realValue);

	                    ELSE
	                      #tempDWord := #statParameter[#tempLoopIndex].dwordValue;
	                    END_IF;

	                    #statReqWriteParameter.data[#tempPointer + 3] := #tempDWord.%B1;
	                    #statReqWriteParameter.data[#tempPointer + 2] := #tempDWord.%B0;
	                    #tempPointer := #tempPointer + 4;  // Points to the next parameter address

	                  #FORMAT_WORD:
	                    IF (#statDatasetType = #DATA_TYPE_DATASET_REAL) OR (#statDatasetType = #DATA_TYPE_SILENT) THEN
	                      #tempDWord := REAL_TO_DWORD(#statParameter[#tempLoopIndex].realValue);

	                    ELSE
	                      #tempDWord := #statParameter[#tempLoopIndex].dwordValue;
	                    END_IF;

	                    #statReqWriteParameter.data[#tempPointer + 3] := #tempDWord.%B0;
	                    #statReqWriteParameter.data[#tempPointer + 2] := #tempDWord.%B1;
	                    #tempPointer := #tempPointer + 4;  // Points to the next parameter address

	                  ELSE
	                    ;
	                END_CASE;
	              END_FOR; // // Creating parameter address
	            END_IF; // #statCmdBusy = FALSE AND #statParameterConfig = TRUE


	            IF (#statFBSubState = #FB_BUSY_WRREC_1) AND (#statError = FALSE) THEN
	              // WRREC command
	              #instWRREC(REQ := TRUE,                                                // Transfer data record
	                         ID := #statHwId,                                                // ID number of the hardware component
	                         INDEX := #statDataRecordNo,                                                    // Data record number
	                         LEN := 0,                                                       // Maximum length of the data record to be transferred in bytes
	                         DONE => #statCmdDone,                                           // Data record was transferred
	                         BUSY => #statCmdBusy,                                           // The writing process is not yet complete
	                         ERROR => #statCmdError,                                         // An error occurred during the writing process
	                         STATUS => #tempCmdStatus,                                       // Status[1] = Error => Status[2] Error Decode + Status[3] Error Code
	                         RECORD := #statReqReadParameter);                               // Data record

	            ELSIF (#statFBSubState = #FB_BUSY_WRREC_2) AND (#statError = FALSE) THEN
	              // WRREC command
	              #instWRREC(REQ := TRUE,                                                // Transfer data record
	                         ID := #statHwId,                                                // ID number of the hardware component
	                         INDEX := #statDataRecordNo,                                                    // Data record number
	                         LEN := 0,                                                       // Maximum length of the data record to be transferred in bytes
	                         DONE => #statCmdDone,                                           // Data record was transferred
	                         BUSY => #statCmdBusy,                                           // The writing process is not yet complete
	                         ERROR => #statCmdError,                                         // An error occurred during the writing process
	                         STATUS => #tempCmdStatus,                                       // Status[1] = Error => Status[2] Error Decode + Status[3] Error Code
	                         RECORD := #statReqWriteParameter);                              // Data record
	            END_IF;


	            // Error occurred
	            IF (#statCmdError = TRUE) AND (#statError = FALSE) THEN
	              // Get the error information from the status information
	              #tempStatusWord.%B0 := #tempCmdStatus.%B1;
	              #tempStatusWord.%B1 := #tempCmdStatus.%B2;

	              // Temporary command status (80A1, 80A7, 80B5, 80C0, 80C1, 80C2, 80C3 oder 80C4) are valid and retry command
	              IF (#tempStatusWord = 16#80A1) OR  // Negative acknowledgment when writing to the module
	                (#tempStatusWord = 16#80A7) OR   // DP slave or module is occupied (temporary error)
	                (#tempStatusWord = 16#80B5) OR   // DP slave or module not ready
	                (#tempStatusWord = 16#80C0) OR   // The data can only be written when the CPU is in STOP mode. Note: this means that writing by the user program is not possible. You can only write the data online with PG/PC.
	                (#tempStatusWord = 16#80C1) OR   // The data of the previous write job on the module for the same data record have not yet been processed by the module.
	                (#tempStatusWord = 16#80C2) OR   // The module is currently processing the maximum possible number of jobs for a CPU.
	                (#tempStatusWord = 16#80C3) OR   // The required operating resources are currently occupied.
	                (#tempStatusWord = 16#80C4) THEN // Internal temporary error. Job could not be executed. Repeat the job. If this error occurs often, check your installation for sources of electrical interference.

	                IF (#statErrorCount >= #MAX_ERROR_COUNT) THEN
	                  #statError := TRUE;
	                  #statStateNumber := #statFBSubState;
	                  #statSubfunctionStatus := #tempStatusWord;
	                  #statStatus := #ERR_WRREC_TEMP_COUNTER;
	                  #statFBState := #FB_ERROR;
	                ELSE
	                  #statErrorCount := #statErrorCount + 1;  // Increment internal error counter
	                  #statFBSubStateOld := #statFBSubState;
	                  #statFBSubState := #FB_BUSY_WAIT;
	                END_IF;
	              ELSE
	                #statError := TRUE;
	                #statStateNumber := #statFBSubState;
	                #statSubfunctionStatus := #tempStatusWord;
	                #statStatus := #ERR_WRREC;
	                #statFBState := #FB_ERROR;
	              END_IF; // Temporary command status (80A1, 80A7, 80B5, 80C0, 80C1, 80C2, 80C3 oder 80C4) are valid and retry command

	            ELSIF (#statCmdBusy = FALSE) AND (#statCmdDone = TRUE) AND (#statError = FALSE) AND (#statFBSubState = #FB_BUSY_WRREC_1) THEN  // Processing completed without errors
	              #statErrorCount := 0;  // V1.5.1 Reset error counter
	              #statFBSubState := #FB_BUSY_RDREC_1; // WRREC completed and continue with RDREC

	            ELSIF (#statCmdBusy = FALSE) AND (#statCmdDone = TRUE) AND (#statError = FALSE) AND (#statFBSubState = #FB_BUSY_WRREC_2) THEN  // Processing completed without errors
	              #statErrorCount := 0;  // V1.5.1 Reset error counter
	              #statFBSubState := #FB_BUSY_RDREC_2; // WRREC completed and continue with RDREC
	              // Clearing the receive buffer
	              #statRespParameter.header := #tempVoidHeader;
	              FOR #tempLoopIndex := 0 TO #LENGTH_READ_TELEGRAM_UPPER_LIM DO
	                #statRespParameter.data[#tempLoopIndex] := 16#00;
	              END_FOR;
	            END_IF; // #statCmdError = TRUE

	          #FB_BUSY_RDREC_1, #FB_BUSY_RDREC_2:  // Reading the values from the drive object

	            // Resets RDREC command
	            IF (#statCmdBusy = FALSE) THEN
	              #instRDREC(REQ := FALSE,
	                         RECORD := #statRespParameter);
	            END_IF;

	            #instRDREC(REQ := TRUE,                                                 // Transfer data record
	                       ID := #statHwId,                                                 // ID number of the hardware component
	                       INDEX := #statDataRecordNo,                                                     // Data record number
	                       MLEN := 0,                                                       // Maximum length in bytes of the data record information to be read
	                       VALID => #tempCmdValid,                                          // New data record was received and is valid
	                       BUSY => #statCmdBusy,                                            // The reading process is not yet complete
	                       ERROR => #statCmdError,                                          // An error occurred during the reading process
	                       STATUS => #tempCmdStatus,                                        // Status[1] = Error => Status[2] Error Decode + Status[3] Error Code
	                       RECORD := #statRespParameter);                                   // Destination area for the data record read


	            // Error occurred
	            IF (#statCmdError = TRUE) AND (#statError = FALSE) THEN
	              // Get the error information from the status information
	              #tempStatusWord.%B0 := #tempCmdStatus.%B1;
	              #tempStatusWord.%B1 := #tempCmdStatus.%B2;

	              // Temporary command status (80A0, 80A7, 80B5, 80C0, 80C1, 80C2, 80C3 oder 80C4) are valid and retry command
	              IF (#tempStatusWord = 16#80A0) OR  // Negative acknowledgment when reading the module
	                (#tempStatusWord = 16#80A7) OR   // DP slave or module is occupied (temporary error)
	                (#tempStatusWord = 16#80B5) OR   // DP slave or module not ready
	                (#tempStatusWord = 16#80C0) OR   // The data can only be written when the CPU is in STOP mode. Note: this means that writing by the user program is not possible. You can only write the data online with PG/PC.
	                (#tempStatusWord = 16#80C1) OR   // The data of the previous write job on the module for the same data record have not yet been processed by the module.
	                (#tempStatusWord = 16#80C2) OR   // The module is currently processing the maximum possible number of jobs for a CPU.
	                (#tempStatusWord = 16#80C3) OR   // The required operating resources are currently occupied.
	                (#tempStatusWord = 16#80C4) THEN // Internal temporary error. Job could not be executed. Repeat the job. If this error occurs often, check your installation for sources of electrical interference.


	                IF (#statErrorCount >= #MAX_ERROR_COUNT) THEN
	                  #statError := TRUE;
	                  #statStateNumber := #statFBSubState;
	                  #statSubfunctionStatus := #tempStatusWord;
	                  #statStatus := #ERR_RDREC_TEMP_COUNTER;
	                  #statFBState := #FB_ERROR;
	                ELSE
	                  #statErrorCount := #statErrorCount + 1;  // Increment internal error counter
	                  #statFBSubStateOld := #statFBSubState;
	                  // V1.3.2. If error 80A0 then should be retry with WRREC command
	                  IF (#tempStatusWord = 16#80A0) AND #statFBSubState = #FB_BUSY_RDREC_1 THEN
	                    #statFBSubStateOld := #FB_BUSY_WRREC_1;
	                  ELSIF (#tempStatusWord = 16#80A0) AND #statFBSubState = #FB_BUSY_RDREC_2 THEN
	                    #statFBSubStateOld := #FB_BUSY_WRREC_2;
	                  END_IF;
	                  #statFBSubState := #FB_BUSY_WAIT;
	                END_IF;
	              ELSE
	                #statError := TRUE;
	                #statStateNumber := #statFBSubState;
	                #statSubfunctionStatus := #tempStatusWord;
	                #statStatus := #ERR_RDREC;
	                #statFBState := #FB_ERROR;
	              END_IF; // Temporary command status (80A0, 80A7, 80B5, 80C0, 80C1, 80C2, 80C3 oder 80C4) are valid and retry command

	              // Error : Reference number of the request does not match with the response reference number
	            ELSIF (#statCmdBusy = FALSE) AND
	              (#statRefNo <> BYTE_TO_INT(#statRespParameter.header.refNo)) AND
	              (#tempCmdValid = TRUE) THEN

	              #statError := TRUE;
	              #statStateNumber := #statFBSubState;
	              #statStatus := #ERR_REFERENCE_NO;
	              #statFBState := #FB_ERROR;

	              // Error : Invalid response from the drive object (reqId: 16#01 - reading parameter successful; 16#81: reading parameter finished with error; 16#02: writing parameter sucessful; 16#82: writing parameter finished with error)
	            ELSIF (#statCmdBusy = FALSE) AND
	              NOT (#statRespParameter.header.reqId = 16#81 OR #statRespParameter.header.reqId = 16#01 OR #statRespParameter.header.reqId = 16#02 OR #statRespParameter.header.reqId = 16#82) AND
	              (#tempCmdValid = TRUE) THEN

	              #statError := TRUE;
	              #statStateNumber := #statFBSubState;
	              #statStatus := #ERR_RESPONSE_ID;
	              #statFBState := #FB_ERROR;

	              // Error : The received number of parameters does not match with the requested number of parameters
	            ELSIF (#statCmdBusy = FALSE) AND
	              (#statCountOfElements <> BYTE_TO_INT(#statRespParameter.header.parameterNo)) AND
	              (#tempCmdValid = TRUE) THEN

	              #statError := TRUE;
	              #statStateNumber := #statFBSubState;
	              #statStatus := #ERR_PARAMETER_NO;
	              #statFBState := #FB_ERROR;

	              // Error : The drive object does not match with the responsed DO
	            ELSIF (#statCmdBusy = FALSE) AND
	              (#statDoId <> #statRespParameter.header.doId) AND
	              (#tempCmdValid = TRUE) THEN

	              #statError := TRUE;
	              #statStateNumber := #statFBSubState;
	              #statStatus := #ERR_DRIVE_OBJECT_NO;
	              #statFBState := #FB_ERROR;

	              // No error occurred during reading parameters
	            ELSIF (#statCmdBusy = FALSE) AND (#tempCmdValid = TRUE) AND (#statError = FALSE) THEN

	              IF (#statFBSubState = #FB_BUSY_RDREC_1) THEN

	                // Analyse of the response buffer
	                #tempPointer := 0;
	                FOR #tempLoopIndex := 0 TO #statCountOfElements - 1 DO
	                  #statParameter[#tempLoopIndex].format := #statRespParameter.data[#tempPointer];  // Format of the parameter

	                  // Format = Error
	                  IF (((BYTE_TO_SINT(#statRespParameter.data[#tempPointer]) > #FORMAT_DOUBLE_WORD) OR
	                    ((BYTE_TO_SINT(#statRespParameter.data[#tempPointer]) > #FORMAT_FLOATING_POINT) AND (BYTE_TO_SINT(#statRespParameter.data[#tempPointer]) < #FORMAT_OCTET_STRING)) OR
	                    ((BYTE_TO_SINT(#statRespParameter.data[#tempPointer]) > #FORMAT_OCTET_STRING) AND (BYTE_TO_SINT(#statRespParameter.data[#tempPointer]) < #FORMAT_TIME_DIFFERENCE)) OR
	                    ((BYTE_TO_SINT(#statRespParameter.data[#tempPointer]) > #FORMAT_TIME_DIFFERENCE) AND (BYTE_TO_SINT(#statRespParameter.data[#tempPointer]) < #FORMAT_BYTE)) OR
	                    (BYTE_TO_SINT(#statRespParameter.data[#tempPointer]) < #FORMAT_INTEGER_8))) AND (BYTE_TO_SINT(#statRespParameter.data[#tempPointer]) <> #FORMAT_ZERO)
	                  THEN

	                    #statParameter[#tempLoopIndex].errorValue := #statRespParameter.data[#tempPointer + 3];
	                    // Points to the next parameter address
	                    #tempPointer := #tempPointer + 6;

	                  ELSE
	                    CASE BYTE_TO_SINT(#statRespParameter.data[#tempPointer]) OF
	                      #FORMAT_INTEGER_8, #FORMAT_UNSIGNED_8, #FORMAT_BYTE, #FORMAT_INTEGER_16, #FORMAT_UNSIGNED_16, #FORMAT_OCTET_STRING, #FORMAT_WORD:
	                        #statParameter[#tempLoopIndex].errorValue := 16#FF; // Sets the error status and diagnostic
	                        #tempPointer := #tempPointer + 4; // Points to the next parameter address

	                      #FORMAT_INTEGER_32, #FORMAT_UNSIGNED_32, #FORMAT_TIME_DIFFERENCE, #FORMAT_FLOATING_POINT, #FORMAT_DOUBLE_WORD:
	                        #statParameter[#tempLoopIndex].errorValue := 16#FF; // Sets the error status and diagnostics
	                        #tempPointer := #tempPointer + 6; // Points to the next parameter address

	                      ELSE
	                        ;
	                    END_CASE;
	                  END_IF; // Format = Error
	                END_FOR; // Analyse of the response buffer

	                #statCmdBusy := FALSE;
	                #statCmdError := FALSE;
	                #statFBState := #FB_BUSY;
	                #statFBSubState := #FB_BUSY_WRREC_2;
	              ELSE

	                // Error occurred during writing process (changing parameter values)
	                IF (#statRespParameter.header.reqId = 16#82) THEN  // reqId: 16#82 (Error occurred during writing paramaters)
	                  #tempPointer := 0;

	                  FOR #tempLoopIndex := 0 TO #statCountOfElements - 1 BY 1 DO
	                    // Parameter error
	                    IF (#statRespParameter.data[#tempPointer] = #FORMAT_ERROR) THEN

	                      #statParameter[#tempLoopIndex].errorValue := #statRespParameter.data[#tempPointer + 3]; // V1.3.2
	                      // Save first parameter error in telegram
	                      IF (#statFirstParameterError = #NO_PARAMETER_ERROR) THEN
	                        #statFirstParameterError := #tempLoopIndex;
	                        #diagnostics.firstParameterError := #statFirstParameterError;
	                        #diagnostics.errorValue := #statParameter[#tempLoopIndex].errorValue; // V1.3.2
	                        #statError := TRUE;
	                        #statStateNumber := #statFBSubState;
	                        #statStatus := #ERR_PARAMETER;
	                        #statFBState := #FB_ERROR;
	                      END_IF;

	                      #tempPointer := #tempPointer + 6;  // Points to the next parameter address

	                      // Parameter without errors
	                    ELSE
	                      #statParameter[#tempLoopIndex].errorValue := 16#FF;
	                      #tempPointer := #tempPointer + 2;
	                    END_IF;

	                    IF (#statDatasetType = #DATA_TYPE_SILENT) THEN
	                      #tempSilentOperationData.dataset[#tempLoopIndex].index := #statParameter[#tempLoopIndex].index;
	                      #tempSilentOperationData.dataset[#tempLoopIndex].parameterNumber := #statParameter[#tempLoopIndex].parameterNo;
	                      #tempSilentOperationData.dataset[#tempLoopIndex].value := #statParameter[#tempLoopIndex].realValue;
	                      #tempSilentOperationData.dataset[#tempLoopIndex].errorValue := #statParameter[#tempLoopIndex].errorValue;

	                    ELSIF (#statDatasetType = #DATA_TYPE_DATASET_REAL) THEN
	                      #tempActualElementReal.errorValue := #statParameter[#tempLoopIndex].errorValue;
	                      #tempActualElementReal.index := #statParameter[#tempLoopIndex].index;
	                      #tempActualElementReal.parameterNumber := #statParameter[#tempLoopIndex].parameterNo;
	                      #tempActualElementReal.value := #statParameter[#tempLoopIndex].realValue;
	                      #tempBlkVariant := MOVE_BLK_VARIANT(SRC := #tempActualElementReal, COUNT := 1, SRC_INDEX := 0, DEST_INDEX := #tempLoopIndex, DEST => #dataset);

	                      // Error occurred during MOVE_BLK_VARIANT command
	                      IF (#tempBlkVariant <> 0) THEN
	                        #statError := TRUE;
	                        #statStateNumber := #statFBState;
	                        #statSubfunctionStatus := INT_TO_WORD(#tempBlkVariant);
	                        #statStatus := #ERR_MOVE_BLK_VARIANT;
	                        #statFBState := #FB_ERROR;
	                        #diagnostics.firstParameterError := #tempLoopIndex;
	                      END_IF;

	                      // LAcycCom_typeDriveDatasetDWord is in use
	                    ELSE
	                      #tempActualElementDWord.errorValue := #statParameter[#tempLoopIndex].errorValue;
	                      #tempActualElementDWord.index := #statParameter[#tempLoopIndex].index;
	                      #tempActualElementDWord.parameterNumber := #statParameter[#tempLoopIndex].parameterNo;
	                      #tempActualElementDWord.value := #statParameter[#tempLoopIndex].dwordValue;
	                      #tempBlkVariant := MOVE_BLK_VARIANT(SRC := #tempActualElementDWord, COUNT := 1, SRC_INDEX := 0, DEST_INDEX := #tempLoopIndex, DEST => #dataset);

	                      // Error occurred during MOVE_BLK_VARIANT command
	                      IF (#tempBlkVariant <> 0) THEN
	                        #statError := TRUE;
	                        #statStateNumber := #statFBState;
	                        #statSubfunctionStatus := INT_TO_WORD(#tempBlkVariant);
	                        #statStatus := #ERR_MOVE_BLK_VARIANT;
	                        #statFBState := #FB_ERROR;
	                        #diagnostics.firstParameterError := #tempLoopIndex;
	                      END_IF;
	                    END_IF;
	                  END_FOR;
	                END_IF; // Error occurred during writing process (changing parameter values)

	                #statCmdBusy := FALSE;
	                #statCmdError := FALSE;
	                #statFBSubState := #FB_BUSY_WRREC_1;

	                // Next state is depending on the FB mode
	                IF (#statWithoutResourceManager = FALSE) AND (#statError = FALSE) THEN
	                  #statStatus := #STATUS_RELEASE;
	                  #statFBState := #FB_RELEASE;

	                ELSIF (#statError = FALSE) THEN
	                  #statStatus := #STATUS_EXECUTION_FINISHED;
	                  #statFBState := #FB_DONE;
	                END_IF; // #statMode = #MODE_WITH_BUFFER_MANAGER
	              END_IF; // #statParameterConfig = TRUE
	            END_IF; // #statCmdError = TRUE

	          #FB_BUSY_WAIT:
	            // Timer for temporary errors
	            #instIECTimer(IN := #statTimerStart,
	                          PT := #TIMER_TEMP_ERROR);

	            #statTimerStart := TRUE;
	            IF (#instIECTimer.Q = TRUE) THEN
	              #statTimerStart := FALSE;
	              #statFBSubState := #statFBSubStateOld;
	            END_IF;

	          ELSE
	            #statError := TRUE;
	            #statStatus := #ERR_UNDEFINED_SUBSTATE;
	            #statStateNumber := #statFBState;
	            #statFBState := #FB_ERROR;
	        END_CASE;

	      ELSE
	        #statError := TRUE;
	        #statStatus := #ERR_COMMAND_TIMEOUT;
	        #statStateNumber := #statFBState;
	        #statFBState := #FB_ERROR;
	      END_IF; // ((#buffer.element[#statAllocatedIndex].enable = TRUE) AND (#statMode = #MODE_WITH_BUFFER_MANAGER)) OR #statMode = #MODE_WITHOUT_BUFFER_MANAGER

	    #FB_RELEASE:
	      // Check buffer index for correctness
	      IF (#statAllocatedIndex < 0) OR (#statAllocatedIndex > "LACYCCOM_BUFFER_ELEMENTS_UPPER_LIM") THEN
	        #statError := TRUE;
	        #statStatus := #ERR_INVALID_BUF_INDEX;
	        #statStateNumber := #statFBState;
	        #statFBState := #FB_ERROR;

	      ELSIF (#requestBuffer.header.lockBuffer = FALSE) THEN // V1.5.1
	        #requestBuffer.header.lockBuffer := TRUE;
	        IF (#requestBuffer.elements[#statAllocatedIndex].state.%X0 = TRUE) THEN
	          #requestBuffer.elements[#statAllocatedIndex].state.%X2 := TRUE;
	        ELSE
	          ;
	        END_IF;
	        #requestBuffer.header.lockBuffer := FALSE;
	        #statStatus := #STATUS_EXECUTION_FINISHED;
	        #statFBState := #FB_DONE;

	      END_IF;

	    ELSE
	      #statError := TRUE;
	      #statStatus := #ERR_UNDEFINED_STATE;
	      #statStateNumber := #statFBState;
	      #statFBState := #FB_ERROR;
	  END_CASE;

	  // If input execute is set during processing
	  IF #statWarningRetriggering = TRUE AND #statError = FALSE THEN
	    #statStatus := #WARN_EXECUTE_SET_DURING_PROCESSING;
	  END_IF;

	END_IF; // #statBusy = TRUE


	//----------------------------------------------------------------------
	// Error handling and write outputs
	//----------------------------------------------------------------------

	// Edge detection
	#statExecuteOld := #tempExecute;

	IF (#statFBState = #FB_ERROR) THEN
	  // Release the allocated element when error occurs
	  IF (#statStateNumber <> #FB_FIRST_CYCLE) AND (#statStateNumber <> #FB_ALLOCATE)
	    AND (#statBusy = TRUE) AND (#statWithoutResourceManager = FALSE)
	  THEN
	    IF #requestBuffer.header.lockBuffer = FALSE THEN // V1.5.1
	      #requestBuffer.header.lockBuffer := TRUE;
	      IF (#requestBuffer.elements[#statAllocatedIndex].state.%X0 = TRUE) THEN
	        #requestBuffer.elements[#statAllocatedIndex].state.%X2 := TRUE;
	      ELSE
	        ;
	      END_IF;
	      #requestBuffer.header.lockBuffer := FALSE;

	      // Write diagnostics
	      #diagnostics.stateNumber := #statStateNumber;
	      #diagnostics.subfunctionStatus := #statSubfunctionStatus;
	      #diagnostics.status := #statStatus;
	      #statBusy := FALSE;
	      #statDone := FALSE;

	    END_IF;

	  ELSE
	    // Write diagnostics
	    #diagnostics.stateNumber := #statStateNumber;
	    #diagnostics.subfunctionStatus := #statSubfunctionStatus;
	    #diagnostics.status := #statStatus;
	    #statBusy := FALSE;
	    #statDone := FALSE;
	  END_IF;

	  // FB finished request
	ELSIF (#statFBState = #FB_DONE) THEN

	  // Output for one cycle minimum
	  IF (#tempExecute = FALSE) AND (#statDone = TRUE) THEN
	    #statDone := FALSE;
	    #statStatus := #STATUS_NO_CALL;
	    #statFBState := #FB_IDLE;
	  ELSE
	    #statDone := TRUE;
	    #statBusy := FALSE;
	  END_IF;
	  // If input execute is set during processing
	  IF #statWarningRetriggering = TRUE THEN
	    #statStatus := #ERR_AMBIGUOUS_FB_CALL;
	    #diagnostics.status := #statStatus;
	    #statError := TRUE;
	    #statDone := FALSE;
	  END_IF;
	END_IF;

	// Write static values to outputs

	IF (TypeOf(#dataset) = TypeOf(#tempDatasetRealValue)) OR (TypeOf(#dataset) = TypeOf(#tempDatasetDWordValue)) THEN
	  ;

	ELSIF (TypeOf(#dataset) = LAcycCom_typeDriveSilentOperation) THEN
	  IF (#tempSilentOperationData.functionBlockCommand = "LACYCCOM_NO_COMMAND") OR (#tempSilentOperationData.functionBlockCommand = "LACYCCOM_WRITE_COMMAND") THEN // 16#00: no command; 16#02: write command
	    #tempSilentOperationData.lifeSignCheckFBWrite := #tempSilentOperationData.lifeSignCheckFBWrite + 1;  // Life sign counter to monitor that the FB is enabled
	    #tempSilentOperationData.error := #statError;
	    #tempSilentOperationData.busy := #statBusy;
	    #tempSilentOperationData.done := #statDone;
	    #tempSilentOperationData.status := #statStatus;
	    #tempBlkVariant := MOVE_BLK_VARIANT(SRC := #tempSilentOperationData, COUNT := 1, SRC_INDEX := 0, DEST_INDEX := 0, DEST => #dataset);

	    // Error occurred during MOVE_BLK_VARIANT command
	    IF (#tempBlkVariant <> 0) THEN
	      #statError := TRUE;
	      #statStateNumber := #statFBState;
	      #statSubfunctionStatus := INT_TO_WORD(#tempBlkVariant);
	      #statStatus := #ERR_MOVE_BLK_VARIANT;
	      #statFBState := #FB_ERROR;
	    END_IF;
	  END_IF;

	ELSE
	  #statError := TRUE;
	  #statStatus := #ERR_INVALID_DATA_TYPE;
	  #statFBState := #FB_ERROR;
	END_IF;

	IF #statBusy = FALSE OR #statError = FALSE
	THEN  // V1.5.1
	  #error := #statError;
	  #status := #statStatus;
	END_IF;

	#busy := #statBusy;
	#done := #statDone;
END_FUNCTION_BLOCK

